DATA_BLOCK "Zne03_DB"
{ S7_Optimized_Access := 'TRUE' }
VERSION : 0.1
NON_RETAIN
"Zne03"

BEGIN

END_DATA_BLOCK

